// TwinCAT 3 PLC project AbstactDataStructures
// ProgramVersion: 3.1.4022.7
// libraries:
//   Tc2_Standard, * (Beckhoff Automation GmbH)
//   Tc2_System, * (Beckhoff Automation GmbH)
//   Tc3_Module, * (Beckhoff Automation GmbH)
// project tree:
//   / PlcTask.TcTTO (not stored)
//   POUs/Linked List/DUTs/ T_DATA_TYPE.TcDUT (not stored), ST_NODE.TcDUT
//   POUs/Linked List/ FB_Linked_List.TcPOU, P_Linked_List_Example.TcPOU
//   POUs/ MAIN.TcPOU
// real-time tasks:
//   TASK PlcTask: cycle T#10ms, priority 20, ADS port 350

// ---- POUs/Linked List/DUTs/ST_NODE.TcDUT
{attribute 'enable_dynamic_creation'}
TYPE ST_NODE :
STRUCT
	Data 	: T_DATA_TYPE;
	pNext 	: POINTER TO ST_NODE := NULL;
END_STRUCT
END_TYPE

// ---- POUs/Linked List/FB_Linked_List.TcPOU
// Operated on linked list of type defined by T_DATA_TYPE Alias 
FUNCTION_BLOCK FB_Linked_List
VAR_INPUT
END_VAR
VAR_OUTPUT
END_VAR
VAR
	pHead :  POINTER TO ST_NODE;
	pTail :  POINTER TO ST_NODE;
END_VAR

// Creates/Adds an node to the end of the list
METHOD Create
VAR_INPUT
	Data : T_DATA_TYPE; // Data to add to new node.
END_VAR
VAR
	pTemp :  POINTER TO ST_NODE;
END_VAR
pTemp := __NEW(ST_NODE); 	// Allocate space in memory for a node.
pTemp^.Data := Data;		// Assign Data to the new node.
pTemp^.pNext := NULL;		// Pointer to next node is NULL.
IF pHead = 0 THEN pHead := pTemp; pTail := pTemp; // If the pointer to the pHead is NULL then give it an address. The pTail address of the first node is the pHead.
ELSE  pTail^.pNext := pTemp; pTail := pTail^.pNext; END_IF // Point previous node's pNext to the address of pTemp and set pTail to pTemp.
END_METHOD

// Empties/Clears/Deletes list
METHOD Empty
VAR
	pTemp : POINTER TO ST_NODE;
END_VAR
pTemp := pHead;
WHILE pTemp <> 0 DO
	pTemp := pTemp^.pNext; Pop();
END_WHILE
END_METHOD

// Initializes or create an empty list
METHOD Init
pHead := NULL;
pTail := NULL;
END_METHOD

// Inserts node at a specific position in the list
METHOD Insert
VAR_INPUT
	Data 		: T_DATA_TYPE; 	// Data to add to new node.
	nPosition 	: UXINT;		// Position to add new node in list.
END_VAR
VAR
	pPrevious 	: POINTER TO ST_NODE;
	pCurrent 	: POINTER TO ST_NODE;
	pTemp 		: POINTER TO ST_NODE;
	i 			: UXINT;
END_VAR
pTemp := __NEW(ST_NODE);
pCurrent := pHead;
FOR i := 1 TO nPosition DO
	pPrevious := pCurrent;
	pCurrent := pPrevious^.pNext;
	END_FOR;
pTemp^.Data := Data;
pPrevious^.pNext := pTemp;
pTemp^.pNext := pCurrent;
END_METHOD

// Deletes/pops a node at the start of the list 
METHOD Pop
VAR
	pTemp : POINTER TO ST_NODE;
END_VAR
pTemp := pHead^.pNext;
__DELETE(pHead);
pHead := pTemp;
END_METHOD

// Adds/pushes a node at the start of the list 
METHOD Push
VAR_INPUT
	Data 	: T_DATA_TYPE;
END_VAR
VAR
	pTemp 	:  POINTER TO ST_NODE;
END_VAR
pTemp := __NEW(ST_NODE); 	// Allocate space in memory for a node.
pTemp^.Data := Data;
pTemp^.pNext := pHead;
pHead := pTemp;
END_METHOD

// Deletes node at a specific position in the list
METHOD Remove
VAR_INPUT
	nPosition 	: UXINT; // Position of node to delete.
END_VAR
VAR
	pPrevious 	: POINTER TO ST_NODE;
	pCurrent 	: POINTER TO ST_NODE;
	i 			: UXINT;
END_VAR
pCurrent := pHead;
FOR i := 2 TO nPosition DO
	pPrevious := pCurrent;
	pCurrent := pCurrent^.pNext;
	END_FOR;
pPrevious^.pNext := pCurrent^.pNext;
__DELETE(pCurrent);
END_METHOD

// Traverse the list to display each node
METHOD Show
VAR_IN_OUT
	aList 		: ARRAY[*] OF T_DATA_TYPE; // Array to display data in list.
END_VAR
VAR
	pCurrent 	:  POINTER TO ST_NODE;
	i 			: DINT;
END_VAR
pCurrent := pHead;
i := LOWER_BOUND(aList, 1);
WHILE pCurrent <> 0 AND i < UPPER_BOUND(aList, 1) DO
	aList[i] := pCurrent^.Data;
	pCurrent := pCurrent^.pNext;
	i := i+1;
END_WHILE
END_METHOD

// Gets size of the list
METHOD Size : UXINT;
VAR
	pTemp 	: POINTER TO ST_NODE;
	i 		: UXINT;
END_VAR
pTemp := pHead;
WHILE pTemp <> 0 DO
	pTemp := pTemp^.pNext; i := i + 1;;
END_WHILE
Size := i;
END_METHOD

END_FUNCTION_BLOCK

// ---- POUs/Linked List/P_Linked_List_Example.TcPOU
PROGRAM P_Linked_List_Example
VAR
	nState 			: BYTE;
	fbLinked_List 	: FB_Linked_List;
	
	nSize 			: ULINT; 	// Dispays size of list after it's created
	nDelete_Size 	: ULINT; 	// Displays size of list after deleting an element.
	nInsert_Size 	: ULINT; 	// Displays size of list after inserting an element.
	
	aArray 			: ARRAY[0..5] OF T_DATA_TYPE; // Displays created list.
	aDelete_Array 	: ARRAY[0..5] OF T_DATA_TYPE; // Displays list after deleting element at a position.
	aInsert_Array	: ARRAY[0..5] OF T_DATA_TYPE; // Displays list after inserting element at a position.
	
	 

END_VAR

CASE nState OF 
	0: // Init list.
		fbLinked_List.Init();
		nState := nState + 1;
		
	1: // Create list, display list and list size
		fbLinked_List.Create(1);
		fbLinked_List.Create(2);
		fbLinked_List.Create(3);
		fbLinked_List.Create(4);
		fbLinked_List.Create(5);
		fbLinked_List.Show(aArray);
		nSize := fbLinked_List.Size();

		nState := nState + 1;			
	
	2: // Remove an elements from the list, display list and the list size
		fbLinked_List.Pop();
		fbLinked_List.Remove(3);
		fbLinked_List.Show(aDelete_Array);
		nDelete_Size := fbLinked_List.Size();
		
		nState := nState + 1;
	
	3: // Insert elements into list, display it and the list size
		fbLinked_List.Push(11);
		fbLinked_List.Insert(14,3);
		fbLinked_List.Show(aInsert_Array);
		nInsert_Size := fbLinked_List.Size();
		
		nState := nState + 1;
		
	4: // Clear list, then finish.
		fbLinked_List.Empty();
		
		nState := nState + 1;
END_CASE

END_PROGRAM

// ---- POUs/MAIN.TcPOU
PROGRAM MAIN
VAR
	nState : BYTE;
	fbLinked_List : FB_Linked_List;
	aArray : ARRAY[0..100] OF T_DATA_TYPE;
END_VAR

 CASE nState OF 
	0: // Runs functions once
		fbLinked_List.Init();
		fbLinked_List.Create(1);
		fbLinked_List.Create(2);
		fbLinked_List.Create(3);
		fbLinked_List.Push(12);
		fbLinked_List.Insert(20,2);
		fbLinked_List.Pop();
		
		
		fbLinked_List.Display(aArray);
		nState := nState + 1;
END_CASE

END_PROGRAM
